FUNCTION_BLOCK FB_ConveyerStop
VAR_INPUT
	Execute : BOOL;
END_VAR
VAR_OUTPUT
	Done : BOOL;
END_VAR
VAR
	fbStop : MC_Stop;
END_VAR

IF Execute THEN
Done := TRUE;	
	fbStop(
		Axis := GVL_Conveyer.ConveyerAxis,
		Execute := Execute
		);

Done := fbStop.Done;

END_IF

END_FUNCTION_BLOCK

(* stored: Version 1.1.0.1, ProductVersion 3.1.4024.11
   POU FB_ConveyerStop: Id {04a982e8-5fd2-40b7-9871-383eed3b678c}, SpecialFunc None *)
